// TIA Portal project "02_TIA_Portal" (V17)

(* hardware
DEVICE "S7-1200 station_1"  S7-1200 Station
   slot 0: "Rack_0"  S7-1200 Rack  Rack  V1.0
   slot 1: "PLC_1"  CPU 1214C DC/DC/DC  6ES7 214-1AG40-0XB0  V4.5
DEVICE "HMI_1"  KTP700 Basic PN Portrait
   slot 0: "HMI_1"  KTP700 Basic PN Portrait  6AV2 123-2GB03-0AX0  17.0.0.0
   slot 1: "HMI_RT_1"  KTP700 Basic PN Portrait  6AV2 123-2GB03-0AX0  17.0.0.0
   slot 5: "HMI_1.IE_CP_1"  PROFINET Interface  17.0.0.0
      slot 1: "PROFINET Interface_1"  PROFINET Interface
         slot 1: "Port_1"  Port
*)

// ===== PLC "PLC_1"  CPU 1214C DC/DC/DC =====

VAR_GLOBAL   // PLC tag table "默认变量表"
   "Clock_Byte" AT %MB0 : Byte;
   "Clock_10Hz" AT %M0.0 : Bool;
   "Clock_5Hz" AT %M0.1 : Bool;
   "Clock_2.5Hz" AT %M0.2 : Bool;
   "Clock_2Hz" AT %M0.3 : Bool;
   "Clock_1.25Hz" AT %M0.4 : Bool;
   "Clock_1Hz" AT %M0.5 : Bool;
   "Clock_0.625Hz" AT %M0.6 : Bool;
   "Clock_0.5Hz" AT %M0.7 : Bool;
   "启动按钮" AT %M10.0 : Bool;
   "关闭按钮" AT %M10.1 : Bool;
   "电机线圈" AT %M10.2 : Bool;
END_VAR

TYPE "Equip_Data"
   STRUCT
      Motor_Status : Bool;
      Motor_Speed : Int;
      Temperature : Real;
      Alarm_Code : Int;
      Cmd_Start : Bool;
      Cmd_Stop : Bool;
   END_STRUCT;
END_TYPE

DATA_BLOCK "Data_Hub"   // DB1
{ S7_Optimized_Access := 'FALSE' }
VERSION : 0.1
   VAR
      Line_1 : "Equip_Data";
      Static_1 : Bool;
   END_VAR
BEGIN
END_DATA_BLOCK

DATA_BLOCK "FB_Equipment_Control_DB"   // DB2
{ S7_Optimized_Access := 'TRUE' }
VERSION : 0.1
// stored: InstanceOfName FB_Equipment_Control
"FB_Equipment_Control"
BEGIN
END_DATA_BLOCK

FUNCTION_BLOCK "FB_Equipment_Control"   // FB1, SCL
{ S7_Optimized_Access := 'TRUE' }
VERSION : 0.1
   VAR_IN_OUT
      Equip : "Equip_Data";
   END_VAR
   VAR
      State_Step : Int;
      Stat_Last_Clock : Bool;
      Timer_Heating : TON_TIME;
   END_VAR
BEGIN
   // ==============================================================================
   // 模块名称：FB_Equipment_Control (设备核心控制功能块)
   // 架构设计：基于有限状态机 (FSM) + 面向对象 (OOP) + 物理孪生仿真
   // 核心机制：严格的指令核销、多重防呆互锁、看门狗超时监控
   // ==============================================================================

   // ==========================================
   // Zone 1：第一道防线（最高优先级硬件防呆与安全互锁）
   // 架构原则：安全逻辑必须在最顶层，且按严重程度自上而下排他执行 (ELSIF)
   // ==========================================
   IF #Equip.Temperature > 200.0 OR #Equip.Temperature < -50.0 THEN
       // [致命故障] 传感器物理断线或短路，读取到极端飞值
       #State_Step := 99;                 // 强行踢入故障锁定档
       #Equip.Alarm_Code := 3;            // 报警码 3：传感器异常
       #Equip.Motor_Status := FALSE;      // 强制切断物理输出

   ELSIF #Equip.Temperature >= 80.0 THEN
       // [严重故障] 极限超温保护
       #State_Step := 99;                 // 强行踢入故障锁定档
       #Equip.Alarm_Code := 2;            // 报警码 2：极限超温停机

   ELSIF #Equip.Temperature > 75.0 AND #State_Step <> 99 THEN
       // [一般警告] 高温预警（仅亮黄灯提示，不打断当前设备的运行状态）
       #Equip.Alarm_Code := 1;            // 报警码 1：高温预警

   ELSE
       // [系统正常] 只有在系统没有被 99 号故障锁定时，才允许亮绿灯
       IF #State_Step <> 99 THEN
           #Equip.Alarm_Code := 0;        // 报警码 0：系统正常
       END_IF;
   END_IF;


   // ==========================================
   // Zone 1.5：人类愚蠢操作互锁（防呆拦截）
   // ==========================================
   // 现场极其常见的误操作：工人由于紧张或手套过厚，同时按下了【启动】和【停止】
   IF #Equip.Cmd_Start = TRUE AND #Equip.Cmd_Stop = TRUE THEN
       #Equip.Cmd_Start := FALSE;         // 毫不犹豫地将启动指令抹杀（停止绝对优先）
   END_IF;


   // ==========================================
   // Zone 2：核心大脑（有限状态机 FSM）
   // 架构原则：设备必须具有明确的生命周期，状态绝对互斥
   // ==========================================
   CASE #State_Step OF

       0:  // 【步序 0：待机档 Idle】
           #Equip.Motor_Status := FALSE;

           // 启动条件：收到启动脉冲 AND 系统无任何报警
           IF #Equip.Cmd_Start = TRUE AND #Equip.Alarm_Code = 0 THEN
               #State_Step := 10;         // 挂入 10 档（开始加热冲刺）
               #Equip.Cmd_Start := FALSE; // [核心] 指令生命周期完结，立即核销
           END_IF;

       10: // 【步序 10：加热冲刺档 Heating】
           #Equip.Motor_Status := TRUE;

           // 目标达成机制：温度升至 60 度标准工作温度
           IF #Equip.Temperature >= 60.0 THEN
               #State_Step := 20;         // 目标达成，切入 20 档（稳定保温），看门狗自动解除！
           END_IF;

           // 随时响应人工停机指令
           IF #Equip.Cmd_Stop = TRUE THEN
               #State_Step := 0;
               #Equip.Cmd_Stop := FALSE;  // [核心] 指令核销
           END_IF;

       20: // 【步序 20：稳定运行/保温档 Running】
           // 设备进入此档位，说明各项参数均已达标，进入长效运行期
           #Equip.Motor_Status := TRUE;

           // 随时响应人工停机指令
           IF #Equip.Cmd_Stop = TRUE THEN
               #State_Step := 0;
               #Equip.Cmd_Stop := FALSE;  // [核心] 指令核销
           END_IF;

       99: // 【步序 99：故障锁定档 Fault】
           #Equip.Motor_Status := FALSE;  // 持续锁定输出

           // 故障复位条件：温度自然冷却至 70 度以下，且人工按下【停止(复位)】按钮
           IF #Equip.Temperature < 70.0 AND #Equip.Cmd_Stop = TRUE THEN
               #State_Step := 0;          // 锁定解除，退回待机档准备下一次生产
               #Equip.Cmd_Stop := FALSE;  // [核心] 复位指令核销
           END_IF;

   END_CASE;

   // 【终极指令清洗】：防止处于报警等非接收状态时，指令堆积导致复位后“幽灵自启”
   #Equip.Cmd_Start := FALSE;


   // ==========================================
   // Zone 3：动作超时看门狗 (Watchdog Timer)
   // 监控对象：加热器物理性能评估
   // ==========================================
   // 设定说明：从 20 度加热到 60 度，物理仿真需 40 秒。设定 PT 为 50 秒。
   // 如果状态机卡在 10 档超过 50 秒，必定是加热管断裂或电机皮带断裂！
   #Timer_Heating(IN := (#State_Step = 10),
                  PT := T#50S);

   IF #Timer_Heating.Q = TRUE THEN
       #State_Step := 99;                 // 强行锁死进入故障档
       #Equip.Alarm_Code := 4;            // 报警码 4：加热超时/物理损坏
       #Equip.Motor_Status := FALSE;
   END_IF;


   // ==========================================
   // Zone 4：物理数字孪生引擎 (Thermodynamics & Motion Sim)
   // 作用：无需真实硬件，在 PLC 内部模拟设备的声光热电反馈
   // ==========================================
   // 依赖全局时钟脉冲 "Clock_1Hz" 进行秒级迭代
   IF "Clock_1Hz" = TRUE AND #Stat_Last_Clock = FALSE THEN

       IF #Equip.Motor_Status = TRUE THEN
           // [做功状态]：电机满载，系统每秒升温
           #Equip.Motor_Speed := 1500;
           #Equip.Temperature := #Equip.Temperature + 1.0;
       ELSE
           // [停机状态]：电机停转，系统遵循牛顿冷却定律散热
           #Equip.Motor_Speed := 0;
           IF #Equip.Temperature > 20.0 THEN
               #Equip.Temperature := #Equip.Temperature - 1.0;
           ELSE
               #Equip.Temperature := 20.0; // 触底环境温度
           END_IF;
       END_IF;

   END_IF;

   // 记忆上一扫描周期的时钟状态（实现沿检测闭环）
   #Stat_Last_Clock := "Clock_1Hz";
END_FUNCTION_BLOCK

ORGANIZATION_BLOCK "Main"   // OB1, LAD, ProgramCycle
TITLE = "Main Program Sweep (Cycle)"
{ S7_Optimized_Access := 'TRUE' }
VERSION : 0.1
   VAR_INPUT
      Initial_Call : Bool;   // Initial call of this OB
      Remanence : Bool;   // =True, if remanent data are available
   END_VAR
BEGIN

REGION Network 1
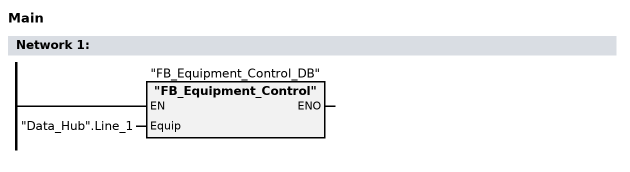
   RUNG wire#powerrail
      "FB_Equipment_Control_DB"(Equip := "Data_Hub".Line_1)
   END_RUNG
   // the same network as SCL:
   "FB_Equipment_Control_DB"(Equip := "Data_Hub".Line_1);   // "FB_Equipment_Control"
END_REGION
END_ORGANIZATION_BLOCK

(* ===== HMI "HMI_RT_1" =====
system functions are stored by id; their names below are inferred from use
connection "HMI_连接_1": ETHERNET, SMART_S7_1200_OMS
connection "HMI_连接_2": ETHERNET, SMART_S7_1200_OMS

HMI tags "默认变量表"
   "Tag_ScreenNumber" : UInt, internal
   "Data_Hub_Line_1_Motor_Status" : Bool = PLC Data_Hub.Line_1.Motor_Status AT %DB1.DBX0.0, 1 s
   "Data_Hub_Line_1_Temperature" : Real = PLC Data_Hub.Line_1.Temperature AT %DB1.DBD4, 1 s
   "Data_Hub_Line_1_Motor_Speed" : Int = PLC Data_Hub.Line_1.Motor_Speed AT %DB1.DBW2, 1 s
   "Data_Hub_Line_1_Alarm_Code" : Int = PLC Data_Hub.Line_1.Alarm_Code AT %DB1.DBW8, 1 s
   "Data_Hub_Line_1_Cmd_Start" : Bool = PLC Data_Hub.Line_1.Cmd_Start AT %DB1.DBX10.0, 1 s
   "Data_Hub_Line_1_Cmd_Stop" : Bool = PLC Data_Hub.Line_1.Cmd_Stop AT %DB1.DBX10.1, 1 s

text list "Alarm_Dict": 0 '系统正常'; 1 '高温预警'; 2 '极限超温停机'; 3 '传感器断线异常'; 4 '加热超时硬件损坏'

Template "模板_1" 480x800
   DateTimeField "HmiScreenItemData" at 375,30 size 105x30
   DateTimeField "HmiScreenItemData_1" at 375,0 size 105x30

screen "根画面" 480x800, template "模板_1"
   on GenerateScreen: SetTag("Tag_ScreenNumber", 1)
   Button "按钮_1" at 14,67 size 166x83; TextOff '启动电机'
      on Press: SetBit("Data_Hub_Line_1_Cmd_Start")
   IOField "I/O 域_1" at 18,226 size 120x64; FormatPattern s99.9
      ProcessValue <- "Data_Hub_Line_1_Temperature"
   IOField "I/O 域_2" at 238,229 size 121x61; FormatPattern s99999
      ProcessValue <- "Data_Hub_Line_1_Motor_Speed"
   TextField "文本域_1" at 54,196 size 39x20; Text '温度'
   TextField "文本域_2" at 279,198 size 39x20; Text '转速'
   SymbolicIOField "符号 I/O 域_1" at 33,316 size 400x428; TextOff '0'; TextOn '1'; TextList "Alarm_Dict"
      ProcessValue <- "Data_Hub_Line_1_Alarm_Code"
      Appearance <- "Data_Hub_Line_1_Alarm_Code"
   Button "按钮_2" at 205,67 size 166x83; TextOff '停止电机'
      on Press: SetBit("Data_Hub_Line_1_Cmd_Stop")
*)